// TIA Portal V17 export
// export: Created 2024-09-02T12:50:02.0436776Z, ExportSetting WithDefaults, DisplayName Totally Integrated Automation Portal, DisplayVersion V17, DisplayName TIA Portal Openness, DisplayVersion V17, DisplayName TIA Portal Version Control Interface, DisplayVersion V17, DisplayName STEP 7 Professional, DisplayVersion V17, DisplayName STEP 7 Safety, DisplayVersion V17, DisplayName WinCC Professional, DisplayVersion V17
FUNCTION_BLOCK "GraFB_Hand_11_20"   // FB1171, GRAPH
TITLE = GRAPH FB
AUTHOR : VAF
FAMILY : SK
NAME : SK
VERSION : 0.1
// Hand functions / Handfunktionen
// stored: AcknowledgeErrorsRequired true, AutoNumber true, ExtensionBlockName LTLL_ManualGraphExt, GraphVersion 4.0, InitialValuesAcquisition false, IsIECCheckEnabled false, LanguageInNetworks LAD, LockOperatingMode false, PermanentILProcessingInMANMode true, SetENOAutomatically false, SkipSteps false, UDAEnableTagReadback false, WithAlarmHandling true
   // inherited from GRAPH_BASE
   VAR
      OFF_SQ_BASE : Bool;
   END_VAR
   VAR_INPUT
      OFF_SQ : Bool;
      INIT_SQ : Bool;
      ACK_EF : Bool;
      S_PREV : Bool;
      S_NEXT : Bool;
      SW_AUTO : Bool;
      SW_TAP : Bool;
      SW_MAN : Bool;
      S_SEL : Int;
      S_ON : Bool;
      S_OFF : Bool;
      T_PUSH : Bool;
   END_VAR
   VAR_OUTPUT
      S_NO : Int;
      S_MORE : Bool;
      S_ACTIVE : Bool;
      ERR_FLT : Bool;
      AUTO_ON : Bool;
      TAP_ON : Bool;
      MAN_ON : Bool;
   END_VAR
   VAR
      extBlock { S7_SetPoint := 'True'} : "LTLL_ManualGraphExt";
   END_VAR
   VAR_TEMP
      t_FrgHand : Bool;   // Freigabe Handbetrieb / Enable manual operation
      t_Service : Bool;   // Servicebetrieb aktiv / Service operation active
   END_VAR
BEGIN
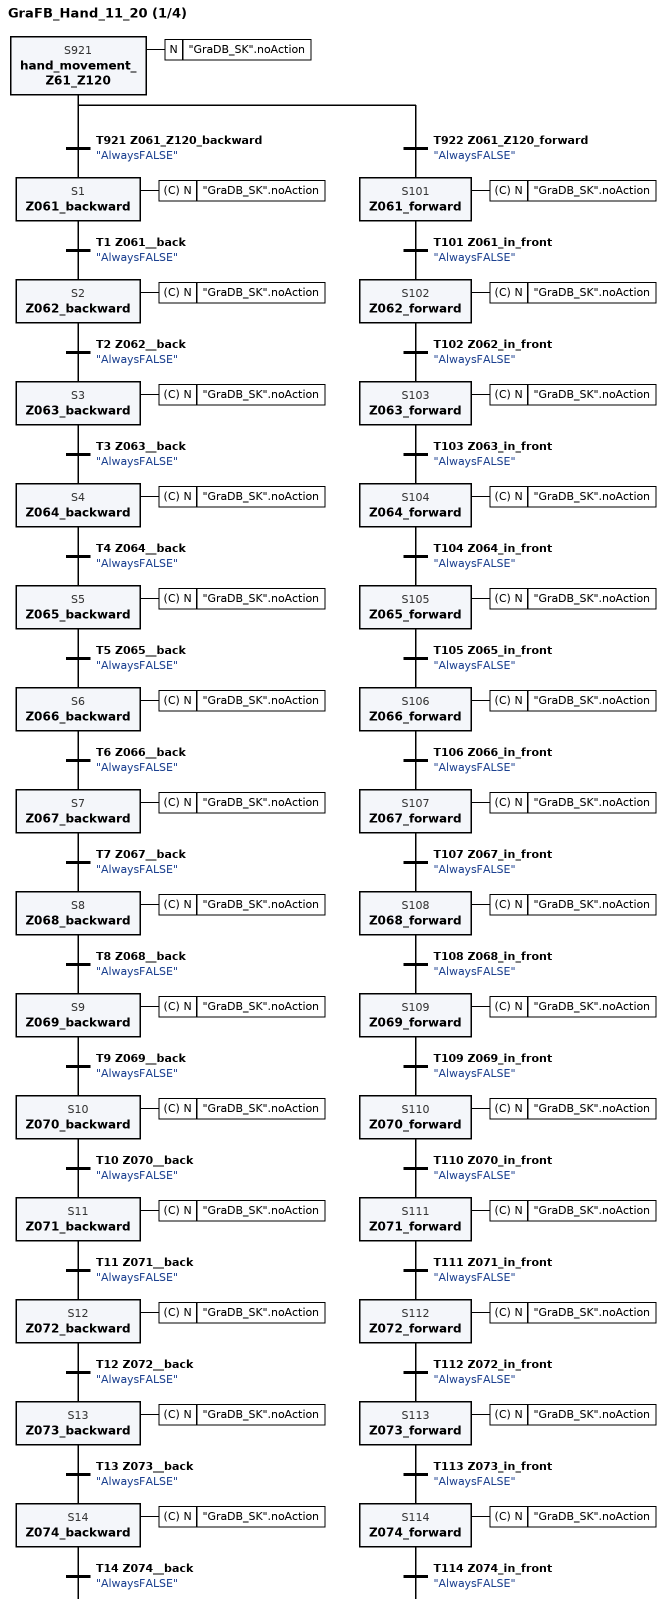
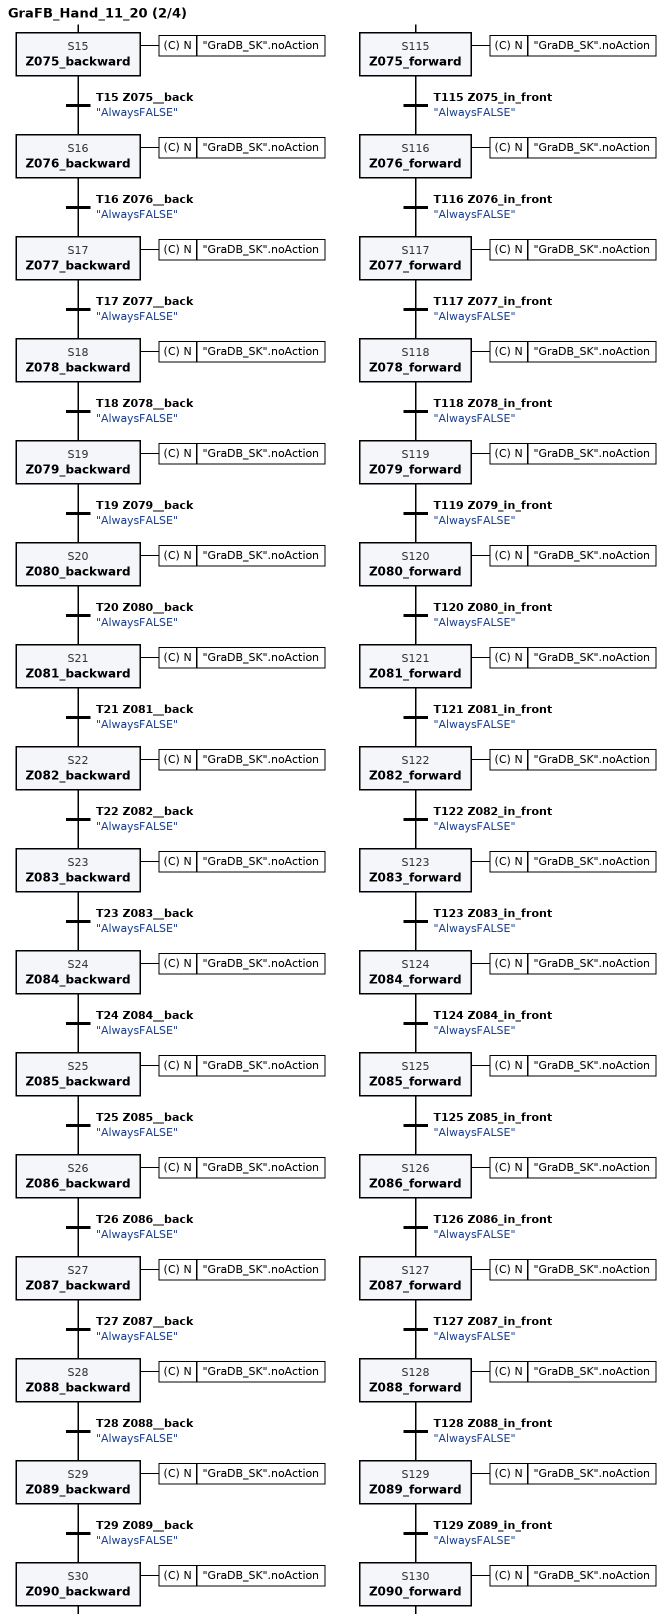
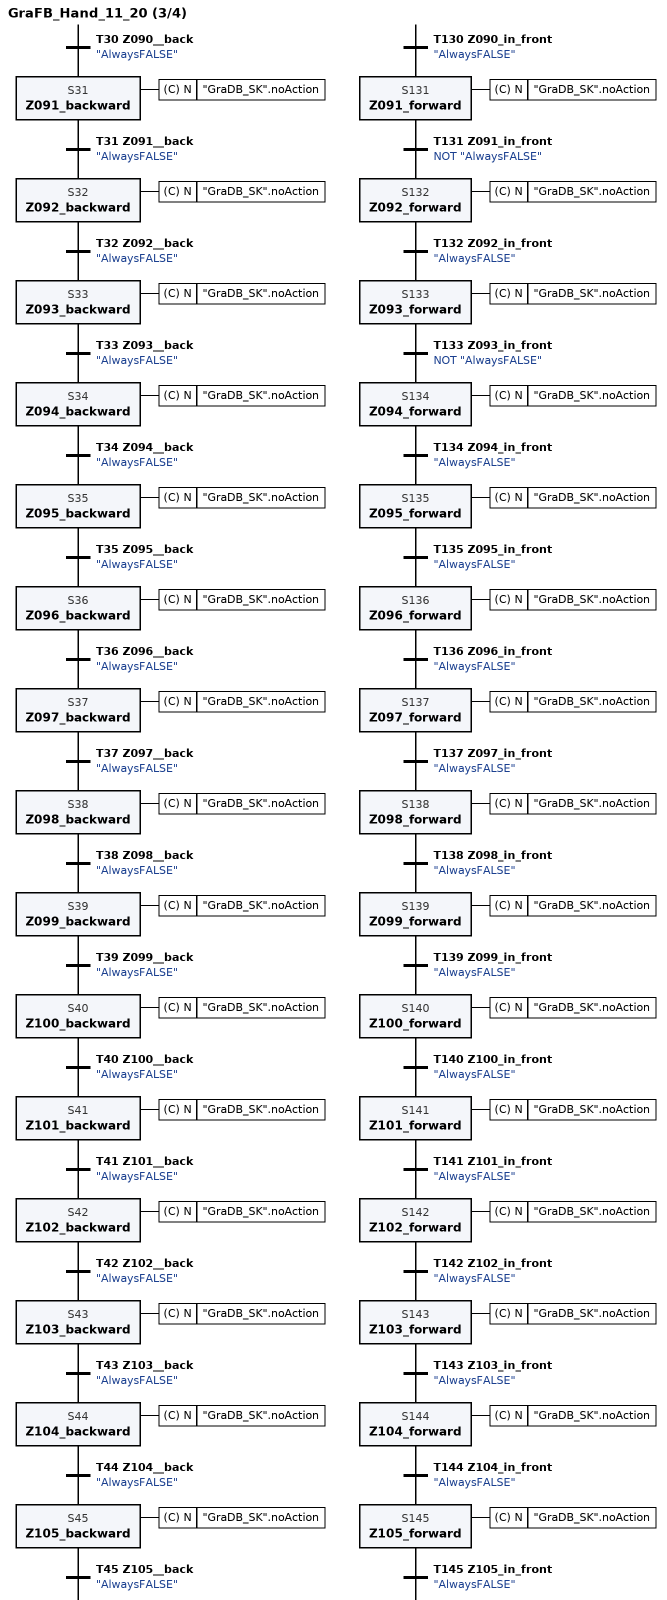
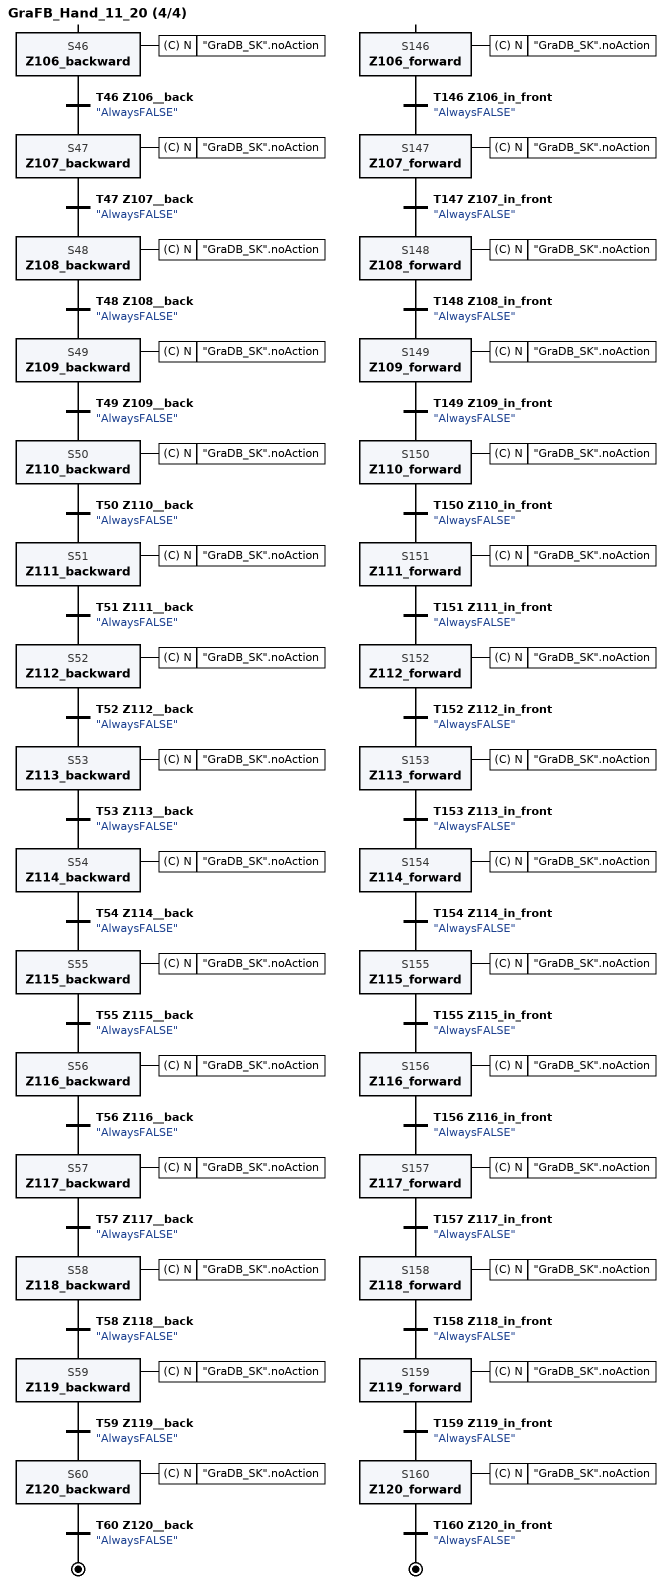
   // permanent pre-instructions
   NETWORK 1
   TITLE = HMI Lite Pass on data / HMI Lite Daten weiterreichen
      #extBlock.input := "LTLL_ManualGraphControl_OP70".screen[0].input;
   NETWORK 2
   TITLE = Instance DB Name query and pass on / Instanz DB Name abfragen und weiterreichen
      GetInstanceName(size := 0, OUT => #extBlock.input.instanceName);
   NETWORK 3
   TITLE = Interlocks Permanent machining, manual Approve and service / Interlocks Permanent Bearbeiten, Handfreigabe und Service
      IF NOT #RT_DATA.MOP.IL_PERM THEN #RT_DATA.MOP.IL_PERM := TRUE; END_IF;
      #t_FrgHand := "AnwDB_OperatingModes_OP70".BA[0]."mode_hand+start";
      #t_Service := "AnwDB_OperatingModes_OP70".BA[0].mode_service;

   // sequencer 1: Sequencer 1
   STEP hand_movement_Z61_Z120:   // S921, max time T#10S, warning time T#7S: Step commentary / Schrittkommentar
      interlock C := (none);   // hand_bereich_Z001_Z005
      supervision V := (none);   // hand_bereich_Z001_Z005
              N    "GraDB_SK".noAction
   END_STEP
   TRANSITION Z061_Z120_backward FROM hand_movement_Z61_Z120 TO Z061_backward   // T921
      := "AlwaysFALSE";
   END_TRANSITION
   TRANSITION Z061_Z120_forward FROM hand_movement_Z61_Z120 TO Z061_forward   // T922
      := "AlwaysFALSE";
   END_TRANSITION
   STEP Z061_backward:   // S1, max time T#10S, warning time T#7S
      interlock C := #t_FrgHand AND ("AlwaysFALSE" OR #t_Service);   // Z061_zur
      supervision V := NOT #Z061__back.TT AND (#Z061_backward.T > T#10S);   // Z061_zur
      (C)     N    "GraDB_SK".noAction
   END_STEP
   TRANSITION Z061__back FROM Z061_backward TO Z062_backward   // T1
      := "AlwaysFALSE";
   END_TRANSITION
   STEP Z062_backward:   // S2, max time T#10S, warning time T#7S
      interlock C := #t_FrgHand AND ("AlwaysFALSE" OR #t_Service);   // Z062_zur
      supervision V := NOT #Z062__back.TT AND (#Z062_backward.T > T#10S);   // Z062_zur
      (C)     N    "GraDB_SK".noAction
   END_STEP
   TRANSITION Z062__back FROM Z062_backward TO Z063_backward   // T2
      := "AlwaysFALSE";
   END_TRANSITION
   STEP Z063_backward:   // S3, max time T#10S, warning time T#7S
      interlock C := #t_FrgHand AND "AlwaysFALSE";   // Z063_zur
      supervision V := NOT #Z063__back.TT AND (#Z063_backward.T > T#10S);   // Z063_zur
      (C)     N    "GraDB_SK".noAction
   END_STEP
   TRANSITION Z063__back FROM Z063_backward TO Z064_backward   // T3
      := "AlwaysFALSE";
   END_TRANSITION
   STEP Z064_backward:   // S4, max time T#10S, warning time T#7S
      interlock C := #t_FrgHand AND ("AlwaysFALSE" OR #t_Service);   // Z064_zur
      supervision V := NOT #Z064__back.TT AND (#Z064_backward.T > T#10s);   // Z064_zur
      (C)     N    "GraDB_SK".noAction
   END_STEP
   TRANSITION Z064__back FROM Z064_backward TO Z065_backward   // T4
      := "AlwaysFALSE";
   END_TRANSITION
   STEP Z065_backward:   // S5, max time T#10S, warning time T#7S
      interlock C := #t_FrgHand AND ("AlwaysFALSE" OR #t_Service);   // Z065_zur
      supervision V := NOT #Z065__back.TT AND (#Z065_backward.T > T#10S);   // Z065_zur
      (C)     N    "GraDB_SK".noAction
   END_STEP
   TRANSITION Z065__back FROM Z065_backward TO Z066_backward   // T5
      := "AlwaysFALSE";
   END_TRANSITION
   STEP Z061_forward:   // S101, max time T#10S, warning time T#7S
      interlock C := #t_FrgHand AND ("AlwaysFALSE" OR #t_Service);   // Z061_vor
      supervision V := NOT #Z061_in_front.TT AND (#Z061_forward.T > T#10S);   // Z061_vor
      (C)     N    "GraDB_SK".noAction
   END_STEP
   TRANSITION Z061_in_front FROM Z061_forward TO Z062_forward   // T101
      := "AlwaysFALSE";
   END_TRANSITION
   STEP Z062_forward:   // S102, max time T#10S, warning time T#7S
      interlock C := #t_FrgHand AND ("AlwaysFALSE" OR #t_Service);   // Z062_vor
      supervision V := NOT #Z062_in_front.TT AND (#Z062_forward.T > T#10S);   // Z062_vor
      (C)     N    "GraDB_SK".noAction
   END_STEP
   TRANSITION Z062_in_front FROM Z062_forward TO Z063_forward   // T102
      := "AlwaysFALSE";
   END_TRANSITION
   STEP Z063_forward:   // S103, max time T#10S, warning time T#7S
      interlock C := #t_FrgHand AND "AlwaysFALSE";   // Z063_vor
      supervision V := NOT #Z063_in_front.TT AND (#Z063_forward.T > T#10S);   // Z063_vor
      (C)     N    "GraDB_SK".noAction
   END_STEP
   TRANSITION Z063_in_front FROM Z063_forward TO Z064_forward   // T103
      := "AlwaysFALSE";
   END_TRANSITION
   STEP Z064_forward:   // S104, max time T#10S, warning time T#7S
      interlock C := #t_FrgHand AND ("AlwaysFALSE" OR #t_Service);   // Z064_vor
      supervision V := NOT #Z064_in_front.TT AND (#Z064_forward.T > T#10S);   // Z064_vor
      (C)     N    "GraDB_SK".noAction
   END_STEP
   TRANSITION Z064_in_front FROM Z064_forward TO Z065_forward   // T104
      := "AlwaysFALSE";
   END_TRANSITION
   STEP Z065_forward:   // S105, max time T#10S, warning time T#7S
      interlock C := #t_FrgHand AND ("AlwaysFALSE" OR #t_Service);   // Z065_vor
      supervision V := NOT #Z065_in_front.TT AND (#Z065_forward.T > T#20S);   // Z065_vor
      (C)     N    "GraDB_SK".noAction
   END_STEP
   TRANSITION Z065_in_front FROM Z065_forward TO Z066_forward   // T105
      := "AlwaysFALSE";
   END_TRANSITION
   STEP Z066_backward:   // S6, max time T#10S, warning time T#7S: Cross transport 2 / Quertransport 2
      interlock C := #t_FrgHand AND ("AlwaysFALSE" OR #t_Service);   // Z066_zur
      supervision V := NOT #Z066__back.TT AND (#Z066_backward.T > T#10S);   // Z066_zur
      (C)     N    "GraDB_SK".noAction
   END_STEP
   TRANSITION Z066__back FROM Z066_backward TO Z067_backward   // T6
      := "AlwaysFALSE";
   END_TRANSITION
   STEP Z067_backward:   // S7, max time T#10S, warning time T#7S
      interlock C := #t_FrgHand AND ("AlwaysFALSE" OR #t_Service);   // Z067_zur
      supervision V := NOT #Z067__back.TT AND (#Z067_backward.T > T#10S);   // Z067_zur
      (C)     N    "GraDB_SK".noAction
   END_STEP
   TRANSITION Z067__back FROM Z067_backward TO Z068_backward   // T7
      := "AlwaysFALSE";
   END_TRANSITION
   STEP Z068_backward:   // S8, max time T#10S, warning time T#7S
      interlock C := #t_FrgHand AND ("AlwaysFALSE" OR #t_Service);   // Z068_zur
      supervision V := NOT #Z068__back.TT AND (#Z068_backward.T > T#10S);   // Z068_zur
      (C)     N    "GraDB_SK".noAction
   END_STEP
   TRANSITION Z068__back FROM Z068_backward TO Z069_backward   // T8
      := "AlwaysFALSE";
   END_TRANSITION
   STEP Z069_backward:   // S9, max time T#10S, warning time T#7S
      interlock C := #t_FrgHand AND ("AlwaysFALSE" OR #t_Service);   // Z069_zur
      supervision V := NOT #Z069__back.TT AND (#Z069_backward.T > T#10S);   // Z069_zur
      (C)     N    "GraDB_SK".noAction
   END_STEP
   TRANSITION Z069__back FROM Z069_backward TO Z070_backward   // T9
      := "AlwaysFALSE";
   END_TRANSITION
   STEP Z070_backward:   // S10, max time T#10S, warning time T#7S
      interlock C := #t_FrgHand AND ("AlwaysFALSE" OR #t_Service);   // Z070_zur
      supervision V := NOT #Z070__back.TT AND (#Z070_backward.T > T#10s);   // Z070_zur
      (C)     N    "GraDB_SK".noAction
   END_STEP
   TRANSITION Z070__back FROM Z070_backward TO Z071_backward   // T10
      := "AlwaysFALSE";
   END_TRANSITION
   STEP Z066_forward:   // S106, max time T#10S, warning time T#7S
      interlock C := #t_FrgHand AND ("AlwaysFALSE" OR #t_Service);   // Z066_vor
      supervision V := NOT #Z066_in_front.TT AND (#Z066_forward.T > T#10S);   // Z066_vor
      (C)     N    "GraDB_SK".noAction
   END_STEP
   TRANSITION Z066_in_front FROM Z066_forward TO Z067_forward   // T106
      := "AlwaysFALSE";
   END_TRANSITION
   STEP Z067_forward:   // S107, max time T#10S, warning time T#7S
      interlock C := #t_FrgHand AND ("AlwaysFALSE" OR #t_Service);   // Z067_vor
      supervision V := NOT #Z067_in_front.TT AND (#Z067_forward.T > T#10S);   // Z067_vor
      (C)     N    "GraDB_SK".noAction
   END_STEP
   TRANSITION Z067_in_front FROM Z067_forward TO Z068_forward   // T107
      := "AlwaysFALSE";
   END_TRANSITION
   STEP Z068_forward:   // S108, max time T#10S, warning time T#7S
      interlock C := #t_FrgHand AND ("AlwaysFALSE" OR #t_Service);   // Z068_vor
      supervision V := NOT #Z068_in_front.TT AND (#Z068_forward.T > T#10S);   // Z068_vor
      (C)     N    "GraDB_SK".noAction
   END_STEP
   TRANSITION Z068_in_front FROM Z068_forward TO Z069_forward   // T108
      := "AlwaysFALSE";
   END_TRANSITION
   STEP Z069_forward:   // S109, max time T#10S, warning time T#7S
      interlock C := #t_FrgHand AND ("AlwaysFALSE" OR #t_Service);   // Z069_vor
      supervision V := NOT #Z069_in_front.TT AND (#Z069_forward.T > T#10S);   // Z069_vor
      (C)     N    "GraDB_SK".noAction
   END_STEP
   TRANSITION Z069_in_front FROM Z069_forward TO Z070_forward   // T109
      := "AlwaysFALSE";
   END_TRANSITION
   STEP Z070_forward:   // S110, max time T#10S, warning time T#7S
      interlock C := #t_FrgHand AND ("AlwaysFALSE" OR #t_Service);   // Z070_vor
      supervision V := NOT #Z070_in_front.TT AND (#Z070_forward.T > T#10S);   // Z070_vor
      (C)     N    "GraDB_SK".noAction
   END_STEP
   TRANSITION Z070_in_front FROM Z070_forward TO Z071_forward   // T110
      := "AlwaysFALSE";
   END_TRANSITION
   STEP Z071_backward:   // S11, max time T#10S, warning time T#7S
      interlock C := #t_FrgHand AND ("AlwaysFALSE" OR #t_Service);   // Z071_zur
      supervision V := NOT #Z071__back.TT AND (#Z071_backward.T > T#10S);   // Z071_zur
      (C)     N    "GraDB_SK".noAction
   END_STEP
   TRANSITION Z071__back FROM Z071_backward TO Z072_backward   // T11
      := "AlwaysFALSE";
   END_TRANSITION
   STEP Z072_backward:   // S12, max time T#10S, warning time T#7S
      interlock C := "AlwaysFALSE";   // Z072_zur
      supervision V := NOT #Z072__back.TT AND (#Z072_backward.T > T#10S);   // Z072_zur
      (C)     N    "GraDB_SK".noAction
   END_STEP
   TRANSITION Z072__back FROM Z072_backward TO Z073_backward   // T12
      := "AlwaysFALSE";
   END_TRANSITION
   STEP Z073_backward:   // S13, max time T#10S, warning time T#7S
      interlock C := #t_FrgHand AND ("AlwaysFALSE" OR #t_Service);   // Z073_zur
      supervision V := NOT #Z073__back.TT AND (#Z073_backward.T > T#15s);   // Z073_zur
      (C)     N    "GraDB_SK".noAction
   END_STEP
   TRANSITION Z073__back FROM Z073_backward TO Z074_backward   // T13
      := "AlwaysFALSE";
   END_TRANSITION
   STEP Z074_backward:   // S14, max time T#10S, warning time T#7S
      interlock C := #t_FrgHand AND ("AlwaysFALSE" OR #t_Service);   // Z075_zur
      supervision V := NOT #Z074__back.TT AND (#Z074_backward.T > T#15s);   // Z075_zur
      (C)     N    "GraDB_SK".noAction
   END_STEP
   TRANSITION Z074__back FROM Z074_backward TO Z075_backward   // T14
      := "AlwaysFALSE";
   END_TRANSITION
   STEP Z075_backward:   // S15, max time T#10S, warning time T#7S
      interlock C := #t_FrgHand AND ("AlwaysFALSE" OR #t_Service);   // Z074_zur
      supervision V := NOT #Z076__back.TT AND (#Z075_backward.T > T#15S);   // Z074_zur
      (C)     N    "GraDB_SK".noAction
   END_STEP
   TRANSITION Z075__back FROM Z075_backward TO Z076_backward   // T15
      := "AlwaysFALSE";
   END_TRANSITION
   STEP Z071_forward:   // S111, max time T#10S, warning time T#7S
      interlock C := #t_FrgHand AND ("AlwaysFALSE" OR #t_Service);   // Z071_vor
      supervision V := NOT #Z071_in_front.TT AND (#Z071_forward.T > T#10S);   // Z071_vor
      (C)     N    "GraDB_SK".noAction
   END_STEP
   TRANSITION Z071_in_front FROM Z071_forward TO Z072_forward   // T111
      := "AlwaysFALSE";
   END_TRANSITION
   STEP Z072_forward:   // S112, max time T#10S, warning time T#7S
      interlock C := "AlwaysFALSE";   // Z072_vor
      supervision V := NOT #Z072_in_front.TT AND (#Z072_forward.T > T#10S);   // Z072_vor
      (C)     N    "GraDB_SK".noAction
   END_STEP
   TRANSITION Z072_in_front FROM Z072_forward TO Z073_forward   // T112
      := "AlwaysFALSE";
   END_TRANSITION
   STEP Z073_forward:   // S113, max time T#10S, warning time T#7S
      interlock C := #t_FrgHand AND ("AlwaysFALSE" OR #t_Service);   // Z073_vor
      supervision V := NOT #Z073_in_front.TT AND (#Z073_forward.T > T#15s);   // Z073_vor
      (C)     N    "GraDB_SK".noAction
   END_STEP
   TRANSITION Z073_in_front FROM Z073_forward TO Z074_forward   // T113
      := "AlwaysFALSE";
   END_TRANSITION
   STEP Z074_forward:   // S114, max time T#10S, warning time T#7S
      interlock C := #t_FrgHand AND ("AlwaysFALSE" OR #t_Service);   // Z075_vor
      supervision V := NOT #Z074_in_front.TT AND (#Z074_forward.T > T#15S);   // Z075_vor
      (C)     N    "GraDB_SK".noAction
   END_STEP
   TRANSITION Z074_in_front FROM Z074_forward TO Z075_forward   // T114
      := "AlwaysFALSE";
   END_TRANSITION
   STEP Z075_forward:   // S115, max time T#10S, warning time T#7S
      interlock C := #t_FrgHand AND ("AlwaysFALSE" OR #t_Service);   // Z074_vor
      supervision V := NOT #Z076_in_front.TT AND (#Z075_forward.T > T#15S);   // Z074_vor
      (C)     N    "GraDB_SK".noAction
   END_STEP
   TRANSITION Z075_in_front FROM Z075_forward TO Z076_forward   // T115
      := "AlwaysFALSE";
   END_TRANSITION
   STEP Z076_backward:   // S16, max time T#10S, warning time T#7S
      interlock C := #t_FrgHand AND ("AlwaysFALSE" OR #t_Service);   // Z076_zur
      supervision V := NOT #Z076__back.TT AND (#Z076_backward.T > T#15S);   // Z076_zur
      (C)     N    "GraDB_SK".noAction
   END_STEP
   TRANSITION Z076__back FROM Z076_backward TO Z077_backward   // T16
      := "AlwaysFALSE";
   END_TRANSITION
   STEP Z077_backward:   // S17, max time T#10S, warning time T#7S
      interlock C := #t_FrgHand AND ("AlwaysFALSE" OR #t_Service);   // Z077_zur
      supervision V := NOT #Z077__back.TT AND (#Z077_backward.T > T#15s);   // Z077_zur
      (C)     N    "GraDB_SK".noAction
   END_STEP
   TRANSITION Z077__back FROM Z077_backward TO Z078_backward   // T17
      := "AlwaysFALSE";
   END_TRANSITION
   STEP Z078_backward:   // S18, max time T#10S, warning time T#7S
      interlock C := "AlwaysFALSE";   // Z078_zur
      supervision V := NOT #Z078__back.TT AND (#Z078_backward.T > T#15S);   // Z078_zur
      (C)     N    "GraDB_SK".noAction
   END_STEP
   TRANSITION Z078__back FROM Z078_backward TO Z079_backward   // T18
      := "AlwaysFALSE";
   END_TRANSITION
   STEP Z079_backward:   // S19, max time T#10S, warning time T#7S
      interlock C := "AlwaysFALSE";   // Z079_zur
      supervision V := NOT #Z079__back.TT AND (#Z079_backward.T > T#15S);   // Z079_zur
      (C)     N    "GraDB_SK".noAction
   END_STEP
   TRANSITION Z079__back FROM Z079_backward TO Z080_backward   // T19
      := "AlwaysFALSE";
   END_TRANSITION
   STEP Z080_backward:   // S20, max time T#10S, warning time T#7S
      interlock C := "AlwaysFALSE";   // Z080_zur
      supervision V := NOT #Z080__back.TT AND (#Z080_backward.T > T#15S);   // Z080_zur
      (C)     N    "GraDB_SK".noAction
   END_STEP
   TRANSITION Z080__back FROM Z080_backward TO Z081_backward   // T20
      := "AlwaysFALSE";
   END_TRANSITION
   STEP Z076_forward:   // S116, max time T#10S, warning time T#7S
      interlock C := #t_FrgHand AND ("AlwaysFALSE" OR #t_Service);   // Z076_vor
      supervision V := NOT #Z076_in_front.TT AND (#Z076_forward.T > T#15s);   // Z076_vor
      (C)     N    "GraDB_SK".noAction
   END_STEP
   TRANSITION Z076_in_front FROM Z076_forward TO Z077_forward   // T116
      := "AlwaysFALSE";
   END_TRANSITION
   STEP Z077_forward:   // S117, max time T#10S, warning time T#7S
      interlock C := #t_FrgHand AND ("AlwaysFALSE" OR #t_Service);   // Z077_vor
      supervision V := NOT #Z077_in_front.TT AND (#Z077_forward.T > T#15s);   // Z077_vor
      (C)     N    "GraDB_SK".noAction
   END_STEP
   TRANSITION Z077_in_front FROM Z077_forward TO Z078_forward   // T117
      := "AlwaysFALSE";
   END_TRANSITION
   STEP Z078_forward:   // S118, max time T#10S, warning time T#7S
      interlock C := "AlwaysFALSE";   // Z078_vor
      supervision V := NOT #Z078_in_front.TT AND (#Z078_forward.T > T#15S);   // Z078_vor
      (C)     N    "GraDB_SK".noAction
   END_STEP
   TRANSITION Z078_in_front FROM Z078_forward TO Z079_forward   // T118
      := "AlwaysFALSE";
   END_TRANSITION
   STEP Z079_forward:   // S119, max time T#10S, warning time T#7S
      interlock C := "AlwaysFALSE";   // Z079_vor
      supervision V := NOT #Z079_in_front.TT AND (#Z079_forward.T > T#15S);   // Z079_vor
      (C)     N    "GraDB_SK".noAction
   END_STEP
   TRANSITION Z079_in_front FROM Z079_forward TO Z080_forward   // T119
      := "AlwaysFALSE";
   END_TRANSITION
   STEP Z080_forward:   // S120, max time T#10S, warning time T#7S
      interlock C := "AlwaysFALSE";   // Z080_vor
      supervision V := NOT #Z080_in_front.TT AND (#Z080_forward.T > T#15S);   // Z080_vor
      (C)     N    "GraDB_SK".noAction
   END_STEP
   TRANSITION Z080_in_front FROM Z080_forward TO Z081_forward   // T120
      := "AlwaysFALSE";
   END_TRANSITION
   STEP Z081_backward:   // S21, max time T#10S, warning time T#7S
      interlock C := "AlwaysFALSE";   // Z081_zur
      supervision V := NOT #Z081__back.TT AND (#Z081_backward.T > T#15S);   // Z081_zur
      (C)     N    "GraDB_SK".noAction
   END_STEP
   TRANSITION Z081__back FROM Z081_backward TO Z082_backward   // T21
      := "AlwaysFALSE";
   END_TRANSITION
   STEP Z082_backward:   // S22, max time T#10S, warning time T#7S
      interlock C := #t_FrgHand AND ("AlwaysTRUE" OR #t_Service) AND "AlwaysFALSE";   // Z082_zur
      supervision V := NOT #Z082__back.TT AND (#Z082_backward.T > T#15S);   // Z082_zur
      (C)     N    "GraDB_SK".noAction
   END_STEP
   TRANSITION Z082__back FROM Z082_backward TO Z083_backward   // T22
      := "AlwaysFALSE";
   END_TRANSITION
   STEP Z083_backward:   // S23, max time T#10S, warning time T#7S
      interlock C := #t_FrgHand AND ("AlwaysTRUE" OR #t_Service) AND "AlwaysFALSE";   // Z083_zur
      supervision V := NOT #Z083__back.TT AND (#Z083_backward.T > T#15S);   // Z083_zur
      (C)     N    "GraDB_SK".noAction
   END_STEP
   TRANSITION Z083__back FROM Z083_backward TO Z084_backward   // T23
      := "AlwaysFALSE";
   END_TRANSITION
   STEP Z084_backward:   // S24, max time T#10S, warning time T#7S
      interlock C := #t_FrgHand AND ("AlwaysTRUE" OR #t_Service) AND "AlwaysFALSE";   // Z084_zur
      supervision V := NOT #Z084__back.TT AND (#Z084_backward.T > T#15S);   // Z084_zur
      (C)     N    "GraDB_SK".noAction
   END_STEP
   TRANSITION Z084__back FROM Z084_backward TO Z085_backward   // T24
      := "AlwaysFALSE";
   END_TRANSITION
   STEP Z085_backward:   // S25, max time T#10S, warning time T#7S
      interlock C := #t_FrgHand AND ("AlwaysFALSE" OR #t_Service);   // Z085_zur
      supervision V := NOT #Z085__back.TT AND (#Z085_backward.T > T#10S);   // Z085_zur
      (C)     N    "GraDB_SK".noAction
   END_STEP
   TRANSITION Z085__back FROM Z085_backward TO Z086_backward   // T25
      := "AlwaysFALSE";
   END_TRANSITION
   STEP Z081_forward:   // S121, max time T#10S, warning time T#7S
      interlock C := "AlwaysFALSE";   // Z081_vor
      supervision V := NOT #Z081_in_front.TT AND (#Z081_forward.T > T#15S);   // Z081_vor
      (C)     N    "GraDB_SK".noAction
   END_STEP
   TRANSITION Z081_in_front FROM Z081_forward TO Z082_forward   // T121
      := "AlwaysFALSE";
   END_TRANSITION
   STEP Z082_forward:   // S122, max time T#10S, warning time T#7S
      interlock C := #t_FrgHand AND ("AlwaysTRUE" OR #t_Service) AND "AlwaysFALSE";   // Z082_vor
      supervision V := NOT #Z082_in_front.TT AND (#Z082_forward.T > T#15S);   // Z082_vor
      (C)     N    "GraDB_SK".noAction
   END_STEP
   TRANSITION Z082_in_front FROM Z082_forward TO Z083_forward   // T122
      := "AlwaysFALSE";
   END_TRANSITION
   STEP Z083_forward:   // S123, max time T#10S, warning time T#7S
      interlock C := #t_FrgHand AND ("AlwaysTRUE" OR #t_Service) AND "AlwaysFALSE";   // Z083_vor
      supervision V := NOT #Z083_in_front.TT AND (#Z083_forward.T > T#15S);   // Z083_vor
      (C)     N    "GraDB_SK".noAction
   END_STEP
   TRANSITION Z083_in_front FROM Z083_forward TO Z084_forward   // T123
      := "AlwaysFALSE";
   END_TRANSITION
   STEP Z084_forward:   // S124, max time T#10S, warning time T#7S
      interlock C := #t_FrgHand AND ("AlwaysTRUE" OR #t_Service) AND "AlwaysFALSE";   // Z084_vor
      supervision V := NOT #Z084_in_front.TT AND (#Z084_forward.T > T#15S);   // Z084_vor
      (C)     N    "GraDB_SK".noAction
   END_STEP
   TRANSITION Z084_in_front FROM Z084_forward TO Z085_forward   // T124
      := "AlwaysFALSE";
   END_TRANSITION
   STEP Z085_forward:   // S125, max time T#10S, warning time T#7S
      interlock C := #t_FrgHand AND ("AlwaysFALSE" OR #t_Service);   // Z085_vor
      supervision V := NOT #Z085_in_front.TT AND (#Z085_forward.T > T#10S);   // Z085_vor
      (C)     N    "GraDB_SK".noAction
   END_STEP
   TRANSITION Z085_in_front FROM Z085_forward TO Z086_forward   // T125
      := "AlwaysFALSE";
   END_TRANSITION
   STEP Z086_backward:   // S26, max time T#10S, warning time T#7S
      interlock C := #t_FrgHand AND ("AlwaysFALSE" OR #t_Service);   // Z086_zur
      supervision V := NOT #Z086__back.TT AND (#Z086_backward.T > T#10S);   // Z086_zur
      (C)     N    "GraDB_SK".noAction
   END_STEP
   TRANSITION Z086__back FROM Z086_backward TO Z087_backward   // T26
      := "AlwaysFALSE";
   END_TRANSITION
   STEP Z087_backward:   // S27, max time T#10S, warning time T#7S
      interlock C := #t_FrgHand AND ("AlwaysFALSE" OR #t_Service);   // Z087_zur
      supervision V := NOT #Z087__back.TT AND (#Z087_backward.T > T#10S);   // Z087_zur
      (C)     N    "GraDB_SK".noAction
   END_STEP
   TRANSITION Z087__back FROM Z087_backward TO Z088_backward   // T27
      := "AlwaysFALSE";
   END_TRANSITION
   STEP Z088_backward:   // S28, max time T#10S, warning time T#7S
      interlock C := #t_FrgHand AND ("AlwaysFALSE" OR #t_Service);   // Z088_zur
      supervision V := NOT #Z088__back.TT AND (#Z088_backward.T > T#10S);   // Z088_zur
      (C)     N    "GraDB_SK".noAction
   END_STEP
   TRANSITION Z088__back FROM Z088_backward TO Z089_backward   // T28
      := "AlwaysFALSE";
   END_TRANSITION
   STEP Z089_backward:   // S29, max time T#10S, warning time T#7S
      interlock C := #t_FrgHand AND ("AlwaysFALSE" OR #t_Service);   // Z089_zur
      supervision V := NOT #Z089__back.TT AND (#Z089_backward.T > T#10S);   // Z089_zur
      (C)     N    "GraDB_SK".noAction
   END_STEP
   TRANSITION Z089__back FROM Z089_backward TO Z090_backward   // T29
      := "AlwaysFALSE";
   END_TRANSITION
   STEP Z090_backward:   // S30, max time T#10S, warning time T#7S
      interlock C := #t_FrgHand AND ("AlwaysFALSE" OR #t_Service);   // Z090_zur
      supervision V := NOT #Z090__back.TT AND (#Z090_backward.T > T#10S);   // Z090_zur
      (C)     N    "GraDB_SK".noAction
   END_STEP
   TRANSITION Z090__back FROM Z090_backward TO Z091_backward   // T30
      := "AlwaysFALSE";
   END_TRANSITION
   STEP Z086_forward:   // S126, max time T#10S, warning time T#7S
      interlock C := #t_FrgHand AND ("AlwaysFALSE" OR #t_Service);   // Z086_vor
      supervision V := NOT #Z086_in_front.TT AND (#Z086_forward.T > T#10S);   // Z086_vor
      (C)     N    "GraDB_SK".noAction
   END_STEP
   TRANSITION Z086_in_front FROM Z086_forward TO Z087_forward   // T126
      := "AlwaysFALSE";
   END_TRANSITION
   STEP Z087_forward:   // S127, max time T#10S, warning time T#7S
      interlock C := #t_FrgHand AND ("AlwaysFALSE" OR #t_Service);   // Z087_vor
      supervision V := NOT #Z087_in_front.TT AND (#Z087_forward.T > T#10S);   // Z087_vor
      (C)     N    "GraDB_SK".noAction
   END_STEP
   TRANSITION Z087_in_front FROM Z087_forward TO Z088_forward   // T127
      := "AlwaysFALSE";
   END_TRANSITION
   STEP Z088_forward:   // S128, max time T#10S, warning time T#7S
      interlock C := #t_FrgHand AND ("AlwaysFALSE" OR #t_Service);   // Z088_vor
      supervision V := NOT #Z088_in_front.TT AND (#Z088_forward.T > T#10S);   // Z088_vor
      (C)     N    "GraDB_SK".noAction
   END_STEP
   TRANSITION Z088_in_front FROM Z088_forward TO Z089_forward   // T128
      := "AlwaysFALSE";
   END_TRANSITION
   STEP Z089_forward:   // S129, max time T#10S, warning time T#7S
      interlock C := #t_FrgHand AND ("AlwaysFALSE" OR #t_Service);   // Z089_vor
      supervision V := NOT #Z089_in_front.TT AND (#Z089_forward.T > T#10S);   // Z089_vor
      (C)     N    "GraDB_SK".noAction
   END_STEP
   TRANSITION Z089_in_front FROM Z089_forward TO Z090_forward   // T129
      := "AlwaysFALSE";
   END_TRANSITION
   STEP Z090_forward:   // S130, max time T#10S, warning time T#7S
      interlock C := #t_FrgHand AND ("AlwaysFALSE" OR #t_Service);   // Z090_vor
      supervision V := NOT #Z090_in_front.TT AND (#Z090_forward.T > T#10S);   // Z090_vor
      (C)     N    "GraDB_SK".noAction
   END_STEP
   TRANSITION Z090_in_front FROM Z090_forward TO Z091_forward   // T130
      := "AlwaysFALSE";
   END_TRANSITION
   STEP Z091_backward:   // S31, max time T#10S, warning time T#7S: Step commentary / Schrittkommentar
      interlock C := #t_FrgHand AND ("AlwaysTRUE" OR #t_Service);   // Z091_zur
      supervision V := NOT #Z091__back.TT AND (#Z091_backward.T > T#10S);   // Z091_zur
      (C)     N    "GraDB_SK".noAction
   END_STEP
   TRANSITION Z091__back FROM Z091_backward TO Z092_backward   // T31
      := "AlwaysFALSE";
   END_TRANSITION
   STEP Z092_backward:   // S32, max time T#10S, warning time T#7S: Step commentary / Schrittkommentar
      interlock C := #t_FrgHand AND ("AlwaysTRUE" OR #t_Service) AND "AlwaysFALSE";   // Z092_zur
      supervision V := NOT #Z092__back.TT AND (#Z092_backward.T > T#10S);   // Z092_zur
      (C)     N    "GraDB_SK".noAction
   END_STEP
   TRANSITION Z092__back FROM Z092_backward TO Z093_backward   // T32
      := "AlwaysFALSE";
   END_TRANSITION
   STEP Z093_backward:   // S33, max time T#10S, warning time T#7S: Step commentary / Schrittkommentar
      interlock C := #t_FrgHand AND ("AlwaysTRUE" OR #t_Service) AND "AlwaysFALSE";   // Z093_zur
      supervision V := NOT #Z093__back.TT AND (#Z093_backward.T > T#10S);   // Z093_zur
      (C)     N    "GraDB_SK".noAction
   END_STEP
   TRANSITION Z093__back FROM Z093_backward TO Z094_backward   // T33
      := "AlwaysFALSE";
   END_TRANSITION
   STEP Z094_backward:   // S34, max time T#10S, warning time T#7S: Step commentary / Schrittkommentar
      interlock C := #t_FrgHand AND ("AlwaysTRUE" OR #t_Service) AND "AlwaysFALSE";   // Z094_zur
      supervision V := NOT #Z094__back.TT AND (#Z094_backward.T > T#10S);   // Z094_zur
      (C)     N    "GraDB_SK".noAction
   END_STEP
   TRANSITION Z094__back FROM Z094_backward TO Z095_backward   // T34
      := "AlwaysFALSE";
   END_TRANSITION
   STEP Z095_backward:   // S35, max time T#10S, warning time T#7S: Step commentary / Schrittkommentar
      interlock C := #t_FrgHand AND ("AlwaysTRUE" OR #t_Service) AND "AlwaysFALSE";   // Z095_zur
      supervision V := NOT #Z095__back.TT AND (#Z095_backward.T > T#10S);   // Z095_zur
      (C)     N    "GraDB_SK".noAction
   END_STEP
   TRANSITION Z095__back FROM Z095_backward TO Z096_backward   // T35
      := "AlwaysFALSE";
   END_TRANSITION
   STEP Z091_forward:   // S131, max time T#10S, warning time T#7S: Step commentary / Schrittkommentar
      interlock C := #t_FrgHand AND ("AlwaysTRUE" OR #t_Service) AND "AlwaysFALSE";   // Z091_vor
      supervision V := NOT #Z091_in_front.TT AND (#Z091_forward.T > T#10S);   // Z091_vor
      (C)     N    "GraDB_SK".noAction
   END_STEP
   TRANSITION Z091_in_front FROM Z091_forward TO Z092_forward   // T131
      := NOT "AlwaysFALSE";
   END_TRANSITION
   STEP Z092_forward:   // S132, max time T#10S, warning time T#7S: Step commentary / Schrittkommentar
      interlock C := #t_FrgHand AND ("AlwaysTRUE" OR #t_Service) AND "AlwaysFALSE";   // Z092_vor
      supervision V := NOT #Z092_in_front.TT AND (#Z092_forward.T > T#10S);   // Z092_vor
      (C)     N    "GraDB_SK".noAction
   END_STEP
   TRANSITION Z092_in_front FROM Z092_forward TO Z093_forward   // T132
      := "AlwaysFALSE";
   END_TRANSITION
   STEP Z093_forward:   // S133, max time T#10S, warning time T#7S: Step commentary / Schrittkommentar
      interlock C := #t_FrgHand AND ("AlwaysTRUE" OR #t_Service) AND "AlwaysFALSE";   // Z093_vor
      supervision V := NOT #Z093_in_front.TT AND (#Z093_forward.T > T#10S);   // Z093_vor
      (C)     N    "GraDB_SK".noAction
   END_STEP
   TRANSITION Z093_in_front FROM Z093_forward TO Z094_forward   // T133
      := NOT "AlwaysFALSE";
   END_TRANSITION
   STEP Z094_forward:   // S134, max time T#10S, warning time T#7S: Step commentary / Schrittkommentar
      interlock C := #t_FrgHand AND ("AlwaysTRUE" OR #t_Service) AND "AlwaysFALSE";   // Z094_vor
      supervision V := NOT #Z094_in_front.TT AND (#Z094_forward.T > T#10S);   // Z094_vor
      (C)     N    "GraDB_SK".noAction
   END_STEP
   TRANSITION Z094_in_front FROM Z094_forward TO Z095_forward   // T134
      := "AlwaysFALSE";
   END_TRANSITION
   STEP Z095_forward:   // S135, max time T#10S, warning time T#7S: Step commentary / Schrittkommentar
      interlock C := #t_FrgHand AND ("AlwaysTRUE" OR #t_Service) AND "AlwaysFALSE";   // Z095_vor
      supervision V := NOT #Z095_in_front.TT AND (#Z095_forward.T > T#10S);   // Z095_vor
      (C)     N    "GraDB_SK".noAction
   END_STEP
   TRANSITION Z095_in_front FROM Z095_forward TO Z096_forward   // T135
      := "AlwaysFALSE";
   END_TRANSITION
   STEP Z096_backward:   // S36, max time T#10S, warning time T#7S: Step commentary / Schrittkommentar
      interlock C := #t_FrgHand AND ("AlwaysTRUE" OR #t_Service) AND "AlwaysFALSE";   // Z096_zur
      supervision V := NOT #Z096__back.TT AND (#Z096_backward.T > T#10S);   // Z096_zur
      (C)     N    "GraDB_SK".noAction
   END_STEP
   TRANSITION Z096__back FROM Z096_backward TO Z097_backward   // T36
      := "AlwaysFALSE";
   END_TRANSITION
   STEP Z097_backward:   // S37, max time T#10S, warning time T#7S: Step commentary / Schrittkommentar
      interlock C := #t_FrgHand AND ("AlwaysTRUE" OR #t_Service) AND "AlwaysFALSE";   // Z097_zur
      supervision V := NOT #Z097__back.TT AND (#Z097_backward.T > T#10S);   // Z097_zur
      (C)     N    "GraDB_SK".noAction
   END_STEP
   TRANSITION Z097__back FROM Z097_backward TO Z098_backward   // T37
      := "AlwaysFALSE";
   END_TRANSITION
   STEP Z098_backward:   // S38, max time T#10S, warning time T#7S: Step commentary / Schrittkommentar
      interlock C := #t_FrgHand AND ("AlwaysTRUE" OR #t_Service) AND "AlwaysFALSE";   // Z098_zur
      supervision V := NOT #Z098__back.TT AND (#Z098_backward.T > T#10S);   // Z098_zur
      (C)     N    "GraDB_SK".noAction
   END_STEP
   TRANSITION Z098__back FROM Z098_backward TO Z099_backward   // T38
      := "AlwaysFALSE";
   END_TRANSITION
   STEP Z099_backward:   // S39, max time T#10S, warning time T#7S: Step commentary / Schrittkommentar
      interlock C := #t_FrgHand AND ("AlwaysTRUE" OR #t_Service) AND "AlwaysFALSE";   // Z099_zur
      supervision V := NOT #Z099__back.TT AND (#Z099_backward.T > T#10S);   // Z099_zur
      (C)     N    "GraDB_SK".noAction
   END_STEP
   TRANSITION Z099__back FROM Z099_backward TO Z100_backward   // T39
      := "AlwaysFALSE";
   END_TRANSITION
   STEP Z100_backward:   // S40, max time T#10S, warning time T#7S: Step commentary / Schrittkommentar
      interlock C := #t_FrgHand AND "AlwaysFALSE";   // Z100_zur
      supervision V := NOT #Z100__back.TT AND (#Z100_backward.T > T#10S);   // Z/100_zur
      (C)     N    "GraDB_SK".noAction
   END_STEP
   TRANSITION Z100__back FROM Z100_backward TO Z101_backward   // T40
      := "AlwaysFALSE";
   END_TRANSITION
   STEP Z096_forward:   // S136, max time T#10S, warning time T#7S: Step commentary / Schrittkommentar
      interlock C := #t_FrgHand AND ("AlwaysTRUE" OR #t_Service) AND "AlwaysFALSE";   // Z096_vor
      supervision V := NOT #Z096_in_front.TT AND (#Z096_forward.T > T#10S);   // Z096_vor
      (C)     N    "GraDB_SK".noAction
   END_STEP
   TRANSITION Z096_in_front FROM Z096_forward TO Z097_forward   // T136
      := "AlwaysFALSE";
   END_TRANSITION
   STEP Z097_forward:   // S137, max time T#10S, warning time T#7S: Step commentary / Schrittkommentar
      interlock C := #t_FrgHand AND ("AlwaysTRUE" OR #t_Service) AND "AlwaysFALSE";   // Z097_vor
      supervision V := NOT #Z097_in_front.TT AND (#Z097_forward.T > T#10S);   // Z097_vor
      (C)     N    "GraDB_SK".noAction
   END_STEP
   TRANSITION Z097_in_front FROM Z097_forward TO Z098_forward   // T137
      := "AlwaysFALSE";
   END_TRANSITION
   STEP Z098_forward:   // S138, max time T#10S, warning time T#7S: Step commentary / Schrittkommentar
      interlock C := #t_FrgHand AND ("AlwaysTRUE" OR #t_Service) AND "AlwaysFALSE";   // Z098_vor
      supervision V := NOT #Z098_in_front.TT AND (#Z098_forward.T > T#10S);   // Z098_vor
      (C)     N    "GraDB_SK".noAction
   END_STEP
   TRANSITION Z098_in_front FROM Z098_forward TO Z099_forward   // T138
      := "AlwaysFALSE";
   END_TRANSITION
   STEP Z099_forward:   // S139, max time T#10S, warning time T#7S: Step commentary / Schrittkommentar
      interlock C := #t_FrgHand AND ("AlwaysTRUE" OR #t_Service) AND "AlwaysFALSE";   // Z099_vor
      supervision V := NOT #Z099_in_front.TT AND (#Z099_forward.T > T#10S);   // Z099_vor
      (C)     N    "GraDB_SK".noAction
   END_STEP
   TRANSITION Z099_in_front FROM Z099_forward TO Z100_forward   // T139
      := "AlwaysFALSE";
   END_TRANSITION
   STEP Z100_forward:   // S140, max time T#10S, warning time T#7S: Step commentary / Schrittkommentar
      interlock C := #t_FrgHand AND "AlwaysFALSE";   // Z100_vor
      supervision V := NOT #Z100_in_front.TT AND (#Z100_forward.T > T#10S);   // Z100_vor
      (C)     N    "GraDB_SK".noAction
   END_STEP
   TRANSITION Z100_in_front FROM Z100_forward TO Z101_forward   // T140
      := "AlwaysFALSE";
   END_TRANSITION
   STEP Z101_backward:   // S41, max time T#10S, warning time T#7S: Step commentary / Schrittkommentar
      interlock C := #t_FrgHand AND "AlwaysFALSE";   // Z101_zur
      supervision V := NOT #Z101__back.TT AND (#Z101_backward.T > T#10S);   // Z101_zur
      (C)     N    "GraDB_SK".noAction
   END_STEP
   TRANSITION Z101__back FROM Z101_backward TO Z102_backward   // T41
      := "AlwaysFALSE";
   END_TRANSITION
   STEP Z102_backward:   // S42, max time T#10S, warning time T#7S: Step commentary / Schrittkommentar
      interlock C := #t_FrgHand AND "AlwaysFALSE";   // Z102_zur
      supervision V := NOT #Z102__back.TT AND (#Z102_backward.T > T#10S);   // Z102_zur
      (C)     N    "GraDB_SK".noAction
   END_STEP
   TRANSITION Z102__back FROM Z102_backward TO Z103_backward   // T42
      := "AlwaysFALSE";
   END_TRANSITION
   STEP Z103_backward:   // S43, max time T#10S, warning time T#7S: Step commentary / Schrittkommentar
      interlock C := #t_FrgHand AND ("AlwaysTRUE" OR #t_Service);   // Z103_zur
      supervision V := NOT #Z103__back.TT AND (#Z103_backward.T > T#15S);   // Z103_zur
      (C)     N    "GraDB_SK".noAction
   END_STEP
   TRANSITION Z103__back FROM Z103_backward TO Z104_backward   // T43
      := "AlwaysFALSE";
   END_TRANSITION
   STEP Z104_backward:   // S44, max time T#10S, warning time T#7S: Step commentary / Schrittkommentar
      interlock C := #t_FrgHand AND "AlwaysFALSE";   // Z104_zur
      supervision V := NOT #Z104__back.TT AND (#Z104_backward.T > T#15S);   // Z104_zur
      (C)     N    "GraDB_SK".noAction
   END_STEP
   TRANSITION Z104__back FROM Z104_backward TO Z105_backward   // T44
      := "AlwaysFALSE";
   END_TRANSITION
   STEP Z105_backward:   // S45, max time T#10S, warning time T#7S: Step commentary / Schrittkommentar
      interlock C := #t_FrgHand AND ("AlwaysTRUE" OR #t_Service);   // Z105_zur
      supervision V := NOT #Z105__back.TT AND (#Z105_backward.T > T#15S);   // Z105_zur
      (C)     N    "GraDB_SK".noAction
   END_STEP
   TRANSITION Z105__back FROM Z105_backward TO Z106_backward   // T45
      := "AlwaysFALSE";
   END_TRANSITION
   STEP Z101_forward:   // S141, max time T#10S, warning time T#7S
      interlock C := #t_FrgHand AND "AlwaysFALSE";   // Z101_vor
      supervision V := NOT #Z101_in_front.TT AND (#Z101_forward.T > T#10S);   // Z101_vor
      (C)     N    "GraDB_SK".noAction
   END_STEP
   TRANSITION Z101_in_front FROM Z101_forward TO Z102_forward   // T141
      := "AlwaysFALSE";
   END_TRANSITION
   STEP Z102_forward:   // S142, max time T#10S, warning time T#7S
      interlock C := #t_FrgHand AND "AlwaysFALSE";   // Z102_vor
      supervision V := NOT #Z102_in_front.TT AND (#Z102_forward.T > T#10S);   // Z102_vor
      (C)     N    "GraDB_SK".noAction
   END_STEP
   TRANSITION Z102_in_front FROM Z102_forward TO Z103_forward   // T142
      := "AlwaysFALSE";
   END_TRANSITION
   STEP Z103_forward:   // S143, max time T#10S, warning time T#7S
      interlock C := #t_FrgHand AND ("AlwaysTRUE" OR #t_Service) AND "AlwaysFALSE";   // Z103_vor
      supervision V := NOT #Z103_in_front.TT AND (#Z103_forward.T > T#15S);   // Z103_vor
      (C)     N    "GraDB_SK".noAction
   END_STEP
   TRANSITION Z103_in_front FROM Z103_forward TO Z104_forward   // T143
      := "AlwaysFALSE";
   END_TRANSITION
   STEP Z104_forward:   // S144, max time T#10S, warning time T#7S
      interlock C := #t_FrgHand AND ("AlwaysTRUE" OR #t_Service) AND "AlwaysFALSE";   // Z104_vor
      supervision V := NOT #Z104_in_front.TT AND (#Z104_forward.T > T#15S);   // Z104_vor
      (C)     N    "GraDB_SK".noAction
   END_STEP
   TRANSITION Z104_in_front FROM Z104_forward TO Z105_forward   // T144
      := "AlwaysFALSE";
   END_TRANSITION
   STEP Z105_forward:   // S145, max time T#10S, warning time T#7S
      interlock C := #t_FrgHand AND ("AlwaysTRUE" OR #t_Service) AND "AlwaysFALSE";   // Z105_vor
      supervision V := NOT #Z105_in_front.TT AND (#Z105_forward.T > T#15S);   // Z105_vor
      (C)     N    "GraDB_SK".noAction
   END_STEP
   TRANSITION Z105_in_front FROM Z105_forward TO Z106_forward   // T145
      := "AlwaysFALSE";
   END_TRANSITION
   STEP Z106_backward:   // S46, max time T#10S, warning time T#7S: Step commentary / Schrittkommentar
      interlock C := #t_FrgHand AND ("AlwaysTRUE" OR #t_Service) AND "AlwaysFALSE";   // Z106_zur
      supervision V := NOT #Z106__back.TT AND (#Z106_backward.T > T#15S);   // Z106_zur
      (C)     N    "GraDB_SK".noAction
   END_STEP
   TRANSITION Z106__back FROM Z106_backward TO Z107_backward   // T46
      := "AlwaysFALSE";
   END_TRANSITION
   STEP Z107_backward:   // S47, max time T#10S, warning time T#7S: Step commentary / Schrittkommentar
      interlock C := #t_FrgHand AND ("AlwaysTRUE" OR #t_Service) AND "AlwaysFALSE";   // Z107_zur
      supervision V := NOT #Z107__back.TT AND (#Z107_backward.T > T#15S);   // Z107_zur
      (C)     N    "GraDB_SK".noAction
   END_STEP
   TRANSITION Z107__back FROM Z107_backward TO Z108_backward   // T47
      := "AlwaysFALSE";
   END_TRANSITION
   STEP Z108_backward:   // S48, max time T#10S, warning time T#7S: Step commentary / Schrittkommentar
      interlock C := #t_FrgHand AND ("AlwaysTRUE" OR #t_Service);   // Z108_zur
      supervision V := NOT #Z108__back.TT AND (#Z108_backward.T > T#15S);   // Z108_zur
      (C)     N    "GraDB_SK".noAction
   END_STEP
   TRANSITION Z108__back FROM Z108_backward TO Z109_backward   // T48
      := "AlwaysFALSE";
   END_TRANSITION
   STEP Z109_backward:   // S49, max time T#10S, warning time T#7S: Step commentary / Schrittkommentar
      interlock C := #t_FrgHand AND ("AlwaysFALSE" OR #t_Service);   // Z109_zur
      supervision V := NOT #Z109__back.TT AND (#Z109_backward.T > T#10S);   // Z109_zur
      (C)     N    "GraDB_SK".noAction
   END_STEP
   TRANSITION Z109__back FROM Z109_backward TO Z110_backward   // T49
      := "AlwaysFALSE";
   END_TRANSITION
   STEP Z110_backward:   // S50, max time T#10S, warning time T#7S: Step commentary / Schrittkommentar
      interlock C := #t_FrgHand AND ("AlwaysFALSE" OR #t_Service);   // Z110_zur
      supervision V := NOT #Z110__back.TT AND (#Z110_backward.T > T#10S);   // Z110_zur
      (C)     N    "GraDB_SK".noAction
   END_STEP
   TRANSITION Z110__back FROM Z110_backward TO Z111_backward   // T50
      := "AlwaysFALSE";
   END_TRANSITION
   STEP Z106_forward:   // S146, max time T#10S, warning time T#7S: Step commentary / Schrittkommentar
      interlock C := #t_FrgHand AND ("AlwaysTRUE" OR #t_Service) AND "AlwaysFALSE";   // Z106_vor
      supervision V := NOT #Z106_in_front.TT AND (#Z106_forward.T > T#15S);   // Z106_vor
      (C)     N    "GraDB_SK".noAction
   END_STEP
   TRANSITION Z106_in_front FROM Z106_forward TO Z107_forward   // T146
      := "AlwaysFALSE";
   END_TRANSITION
   STEP Z107_forward:   // S147, max time T#10S, warning time T#7S: Step commentary / Schrittkommentar
      interlock C := #t_FrgHand AND ("AlwaysTRUE" OR #t_Service) AND "AlwaysFALSE";   // Z107_vor
      supervision V := NOT #Z107_in_front.TT AND (#Z107_forward.T > T#15S);   // Z107_vor
      (C)     N    "GraDB_SK".noAction
   END_STEP
   TRANSITION Z107_in_front FROM Z107_forward TO Z108_forward   // T147
      := "AlwaysFALSE";
   END_TRANSITION
   STEP Z108_forward:   // S148, max time T#10S, warning time T#7S: Step commentary / Schrittkommentar
      interlock C := #t_FrgHand AND ("AlwaysTRUE" OR #t_Service) AND "AlwaysFALSE";   // Z108_vor
      supervision V := NOT #Z108_in_front.TT AND (#Z108_forward.T > T#15S);   // Z108_vor
      (C)     N    "GraDB_SK".noAction
   END_STEP
   TRANSITION Z108_in_front FROM Z108_forward TO Z109_forward   // T148
      := "AlwaysFALSE";
   END_TRANSITION
   STEP Z109_forward:   // S149, max time T#10S, warning time T#7S: Step commentary / Schrittkommentar
      interlock C := #t_FrgHand AND ("AlwaysFALSE" OR #t_Service);   // Z109_vor
      supervision V := NOT #Z109_in_front.TT AND (#Z109_forward.T > T#10S);   // Z109_vor
      (C)     N    "GraDB_SK".noAction
   END_STEP
   TRANSITION Z109_in_front FROM Z109_forward TO Z110_forward   // T149
      := "AlwaysFALSE";
   END_TRANSITION
   STEP Z110_forward:   // S150, max time T#10S, warning time T#7S: Step commentary / Schrittkommentar
      interlock C := #t_FrgHand AND ("AlwaysFALSE" OR #t_Service);   // Z110_vor
      supervision V := NOT #Z110_in_front.TT AND (#Z110_forward.T > T#10S);   // Z110_vor
      (C)     N    "GraDB_SK".noAction
   END_STEP
   TRANSITION Z110_in_front FROM Z110_forward TO Z111_forward   // T150
      := "AlwaysFALSE";
   END_TRANSITION
   STEP Z111_backward:   // S51, max time T#10S, warning time T#7S: Step commentary / Schrittkommentar
      interlock C := #t_FrgHand AND ("AlwaysFALSE" OR #t_Service);   // Z111_zur
      supervision V := NOT #Z111__back.TT AND (#Z111_backward.T > T#10S);   // Z111_zur
      (C)     N    "GraDB_SK".noAction
   END_STEP
   TRANSITION Z111__back FROM Z111_backward TO Z112_backward   // T51
      := "AlwaysFALSE";
   END_TRANSITION
   STEP Z112_backward:   // S52, max time T#10S, warning time T#7S: Step commentary / Schrittkommentar
      interlock C := #t_FrgHand AND ("AlwaysFALSE" OR #t_Service);   // Z112_zur
      supervision V := NOT #Z112__back.TT AND (#Z112_backward.T > T#10S);   // Z112_zur
      (C)     N    "GraDB_SK".noAction
   END_STEP
   TRANSITION Z112__back FROM Z112_backward TO Z113_backward   // T52
      := "AlwaysFALSE";
   END_TRANSITION
   STEP Z113_backward:   // S53, max time T#10S, warning time T#7S: Step commentary / Schrittkommentar
      interlock C := #t_FrgHand AND ("AlwaysFALSE" OR #t_Service);   // Z113_zur
      supervision V := NOT #Z113__back.TT AND (#Z113_backward.T > T#10S);   // Z113_zur
      (C)     N    "GraDB_SK".noAction
   END_STEP
   TRANSITION Z113__back FROM Z113_backward TO Z114_backward   // T53
      := "AlwaysFALSE";
   END_TRANSITION
   STEP Z114_backward:   // S54, max time T#10S, warning time T#7S: Step commentary / Schrittkommentar
      interlock C := #t_FrgHand AND ("AlwaysFALSE" OR #t_Service);   // Z114_zur
      supervision V := NOT #Z114__back.TT AND (#Z114_backward.T > T#10S);   // Z114_zur
      (C)     N    "GraDB_SK".noAction
   END_STEP
   TRANSITION Z114__back FROM Z114_backward TO Z115_backward   // T54
      := "AlwaysFALSE";
   END_TRANSITION
   STEP Z115_backward:   // S55, max time T#10S, warning time T#7S: Step commentary / Schrittkommentar
      interlock C := #t_FrgHand AND ("AlwaysFALSE" OR #t_Service);   // Z115_zur
      supervision V := NOT #Z115__back.TT AND (#Z115_backward.T > T#10S);   // Z115_zur
      (C)     N    "GraDB_SK".noAction
   END_STEP
   TRANSITION Z115__back FROM Z115_backward TO Z116_backward   // T55
      := "AlwaysFALSE";
   END_TRANSITION
   STEP Z116_backward:   // S56, max time T#10S, warning time T#7S: Step commentary / Schrittkommentar
      interlock C := #t_FrgHand AND ("AlwaysFALSE" OR #t_Service);   // Z116_zur
      supervision V := NOT #Z116__back.TT AND (#Z116_backward.T > T#10S);   // Z116_zur
      (C)     N    "GraDB_SK".noAction
   END_STEP
   TRANSITION Z116__back FROM Z116_backward TO Z117_backward   // T56
      := "AlwaysFALSE";
   END_TRANSITION
   STEP Z117_backward:   // S57, max time T#10S, warning time T#7S: Step commentary / Schrittkommentar
      interlock C := #t_FrgHand AND ("AlwaysFALSE" OR #t_Service);   // Z117_zur
      supervision V := NOT #Z117__back.TT AND (#Z117_backward.T > T#10S);   // Z117_zur
      (C)     N    "GraDB_SK".noAction
   END_STEP
   TRANSITION Z117__back FROM Z117_backward TO Z118_backward   // T57
      := "AlwaysFALSE";
   END_TRANSITION
   STEP Z118_backward:   // S58, max time T#10S, warning time T#7S: Step commentary / Schrittkommentar
      interlock C := #t_FrgHand AND ("AlwaysFALSE" OR #t_Service);   // Z118_zur
      supervision V := NOT #Z118__back.TT AND (#Z118_backward.T > T#10S);   // Z118_zur
      (C)     N    "GraDB_SK".noAction
   END_STEP
   TRANSITION Z118__back FROM Z118_backward TO Z119_backward   // T58
      := "AlwaysFALSE";
   END_TRANSITION
   STEP Z119_backward:   // S59, max time T#10S, warning time T#7S: Step commentary / Schrittkommentar
      interlock C := #t_FrgHand AND ("AlwaysFALSE" OR #t_Service);   // Z119_zur
      supervision V := NOT #Z119__back.TT AND (#Z119_backward.T > T#10S);   // Z119_zur
      (C)     N    "GraDB_SK".noAction
   END_STEP
   TRANSITION Z119__back FROM Z119_backward TO Z120_backward   // T59
      := "AlwaysFALSE";
   END_TRANSITION
   STEP Z120_backward:   // S60, max time T#10S, warning time T#7S: Step commentary / Schrittkommentar
      interlock C := #t_FrgHand AND ("AlwaysFALSE" OR #t_Service);   // Z120_zur
      supervision V := NOT #Z120__back.TT AND (#Z120_backward.T > T#10S);   // Z120_zur
      (C)     N    "GraDB_SK".noAction
   END_STEP
   TRANSITION Z120__back FROM Z120_backward TO END   // T60
      := "AlwaysFALSE";
   END_TRANSITION
   STEP Z111_forward:   // S151, max time T#10S, warning time T#7S
      interlock C := #t_FrgHand AND ("AlwaysFALSE" OR #t_Service);   // Z111_vor
      supervision V := NOT #Z111_in_front.TT AND (#Z111_forward.T > T#10S);   // Z111_vor
      (C)     N    "GraDB_SK".noAction
   END_STEP
   TRANSITION Z111_in_front FROM Z111_forward TO Z112_forward   // T151
      := "AlwaysFALSE";
   END_TRANSITION
   STEP Z112_forward:   // S152, max time T#10S, warning time T#7S
      interlock C := #t_FrgHand AND ("AlwaysFALSE" OR #t_Service);   // Z112_vor
      supervision V := NOT #Z112_in_front.TT AND (#Z112_forward.T > T#10S);   // Z112_vor
      (C)     N    "GraDB_SK".noAction
   END_STEP
   TRANSITION Z112_in_front FROM Z112_forward TO Z113_forward   // T152
      := "AlwaysFALSE";
   END_TRANSITION
   STEP Z113_forward:   // S153, max time T#10S, warning time T#7S
      interlock C := #t_FrgHand AND ("AlwaysFALSE" OR #t_Service);   // Z113_vor
      supervision V := NOT #Z113_in_front.TT AND (#Z113_forward.T > T#10S);   // Z113_vor
      (C)     N    "GraDB_SK".noAction
   END_STEP
   TRANSITION Z113_in_front FROM Z113_forward TO Z114_forward   // T153
      := "AlwaysFALSE";
   END_TRANSITION
   STEP Z114_forward:   // S154, max time T#10S, warning time T#7S
      interlock C := #t_FrgHand AND ("AlwaysFALSE" OR #t_Service);   // Z114_vor
      supervision V := NOT #Z114_in_front.TT AND (#Z114_forward.T > T#10S);   // Z114_vor
      (C)     N    "GraDB_SK".noAction
   END_STEP
   TRANSITION Z114_in_front FROM Z114_forward TO Z115_forward   // T154
      := "AlwaysFALSE";
   END_TRANSITION
   STEP Z115_forward:   // S155, max time T#10S, warning time T#7S
      interlock C := #t_FrgHand AND ("AlwaysFALSE" OR #t_Service);   // Z115_vor
      supervision V := NOT #Z115_in_front.TT AND (#Z115_forward.T > T#10S);   // Z115_vor
      (C)     N    "GraDB_SK".noAction
   END_STEP
   TRANSITION Z115_in_front FROM Z115_forward TO Z116_forward   // T155
      := "AlwaysFALSE";
   END_TRANSITION
   STEP Z116_forward:   // S156, max time T#10S, warning time T#7S: Step commentary / Schrittkommentar
      interlock C := #t_FrgHand AND ("AlwaysFALSE" OR #t_Service);   // Z116_vor
      supervision V := NOT #Z116_in_front.TT AND (#Z116_forward.T > T#10S);   // Z116_vor
      (C)     N    "GraDB_SK".noAction
   END_STEP
   TRANSITION Z116_in_front FROM Z116_forward TO Z117_forward   // T156
      := "AlwaysFALSE";
   END_TRANSITION
   STEP Z117_forward:   // S157, max time T#10S, warning time T#7S: Step commentary / Schrittkommentar
      interlock C := #t_FrgHand AND ("AlwaysFALSE" OR #t_Service);   // Z117_vor
      supervision V := NOT #Z117_in_front.TT AND (#Z117_forward.T > T#10S);   // Z117_vor
      (C)     N    "GraDB_SK".noAction
   END_STEP
   TRANSITION Z117_in_front FROM Z117_forward TO Z118_forward   // T157
      := "AlwaysFALSE";
   END_TRANSITION
   STEP Z118_forward:   // S158, max time T#10S, warning time T#7S: Step commentary / Schrittkommentar
      interlock C := #t_FrgHand AND ("AlwaysFALSE" OR #t_Service);   // Z118_vor
      supervision V := NOT #Z118_in_front.TT AND (#Z118_forward.T > T#10S);   // Z118_vor
      (C)     N    "GraDB_SK".noAction
   END_STEP
   TRANSITION Z118_in_front FROM Z118_forward TO Z119_forward   // T158
      := "AlwaysFALSE";
   END_TRANSITION
   STEP Z119_forward:   // S159, max time T#10S, warning time T#7S: Step commentary / Schrittkommentar
      interlock C := #t_FrgHand AND ("AlwaysFALSE" OR #t_Service);   // Z119_vor
      supervision V := NOT #Z119_in_front.TT AND (#Z119_forward.T > T#10S);   // Z119_vor
      (C)     N    "GraDB_SK".noAction
   END_STEP
   TRANSITION Z119_in_front FROM Z119_forward TO Z120_forward   // T159
      := "AlwaysFALSE";
   END_TRANSITION
   STEP Z120_forward:   // S160, max time T#10S, warning time T#7S: Step commentary / Schrittkommentar
      interlock C := #t_FrgHand AND ("AlwaysFALSE" OR #t_Service);   // Z120_vor
      supervision V := NOT #Z120_in_front.TT AND (#Z120_forward.T > T#10S);   // Z120_vor
      (C)     N    "GraDB_SK".noAction
   END_STEP
   TRANSITION Z120_in_front FROM Z120_forward TO END   // T160
      := "AlwaysFALSE";
   END_TRANSITION

   // permanent post-instructions
   NETWORK 1
   TITLE = HMI Lite Pass on data / HMI Lite Daten weiterreichen
      "LTLL_ManualGraphInterlock"(ManualGraphExtOutput := #extBlock.output,
                              ManualGraphControlScreen := "LTLL_ManualGraphControl_OP70".screen[0]);
   NETWORK 2
   TITLE = Report step error / Schrittkettenfehler melden
      "SysFC_NumOfSQErrors"(FLT := #RT_DATA.SQ_FLAGS.ERR_FLT,
                            Fault_SQ := "AnwDB_OperatingModes_OP70".BA[0].error_report_SK,
                            NumOf_Fault_SQ := "AnwDB_ZP_Alarm_OP70".FaultsNoSK_ST1);
END_FUNCTION_BLOCK
